// Hauptsimulation
CASE nSimulationStep OF
    0: // Initialisierung
        InitializeSimulation();
        nSimulationStep := 10;
        
    10: // Warte auf Start
        Q_bGrdstlgSchrEinh := TRUE;
        Q_bZustellZylAusgef := FALSE;
        fTiefe := 80.0; // Startposition oben
        
        IF I_bSchraubHub THEN
            nSimulationStep := 20;
            Q_sDebugInfo := 'Zylinder fährt aus';
        END_IF
        
    20: // Zylinder ausfahren
        SimulateZylinder();
        
        IF Q_bZustellZylAusgef THEN
            nSimulationStep := 30;
            Q_sDebugInfo := 'Bereit zum Schrauben';
        END_IF
        
    30: // Schraubvorgang simulieren
        SimulateScrewing();
        
        // Zurück wenn Schraubhub weg
        IF NOT I_bSchraubHub THEN
            nSimulationStep := 40;
        END_IF
        
    40: // Rückfahrt
        SimulateRetraction();
        
        IF Q_bGrdstlgSchrEinh THEN
            nSimulationStep := 10;
        END_IF
END_CASE

// NC-Achsen Simulation updaten
UpdateNCAxes();

// Debug-Ausgänge
Q_fSimTiefe := fTiefe;
Q_fSimDrehmoment := fDrehmoment;
Q_fSimDrehzahl := fDrehzahl;

METHOD PRIVATE CalculateRamp : LREAL
VAR_INPUT
    fActual     : LREAL;    // Aktueller Wert
    fTarget     : LREAL;    // Zielwert
    fRampUp     : LREAL;    // Anstiegsgeschwindigkeit
    fRampDown   : LREAL;    // Abstiegsgeschwindigkeit
END_VAR
// Einfache Rampenberechnung
IF fActual < fTarget THEN
    // Aufwärts
    CalculateRamp := fActual + fRampUp;
    IF CalculateRamp > fTarget THEN
        CalculateRamp := fTarget;
    END_IF
ELSIF fActual > fTarget THEN
    // Abwärts
    CalculateRamp := fActual - fRampDown;
    IF CalculateRamp < fTarget THEN
        CalculateRamp := fTarget;
    END_IF
ELSE
    // Ziel erreicht
    CalculateRamp := fTarget;
END_IF

// Begrenzung auf positive Werte
IF CalculateRamp < 0 THEN
    CalculateRamp := 0;
END_IF
END_METHOD

METHOD InitializeSimulation
VAR
END_VAR
// Simulationsparameter basierend auf gewähltem Fall setzen
CASE I_nSimulatedCase OF
    0: // Normalfall - alles OK
        bSchraubeVorhanden := TRUE;
        bMaterialHart := FALSE;
        bMaterialWeich := FALSE;
        Q_sDebugInfo := 'Simulation: Normalfall';
        
    1: // Fall 1: Negative Toleranz & Drehmoment erreicht
        bSchraubeVorhanden := TRUE;
        bMaterialHart := TRUE;
        bMaterialWeich := FALSE;
        Q_sDebugInfo := 'Simulation: Fall 1 - Hartes Material';
        
    2: // Fall 2: Negative Toleranz & Solltiefe erreicht
        bSchraubeVorhanden := TRUE;
        bMaterialHart := FALSE;
        bMaterialWeich := TRUE;
        Q_sDebugInfo := 'Simulation: Fall 2 - Weiches Material';
        
    3: // Fall 3: Positive Toleranz
        bSchraubeVorhanden := TRUE;
        bMaterialHart := FALSE;
        bMaterialWeich := FALSE;
        Q_sDebugInfo := 'Simulation: Fall 3 - Positive Toleranz';
        
    4: // Fall 4: Keine Schraube
        bSchraubeVorhanden := FALSE;
        bMaterialHart := FALSE;
        bMaterialWeich := FALSE;
        Q_sDebugInfo := 'Simulation: Fall 4 - Keine Schraube';
END_CASE

// Startwerte setzen
fAchsPosition := 0;
fTiefe := 80.0; // Startposition oben
fDrehmoment := 0;
fDrehzahl := 0;
fDrehzahlRampe := 0;
fDrehmomentRampe := 0;

// Rampenparameter setzen
fRampeBeschleunigung := 50.0;  // 50 U/min pro 10ms Zyklus = 5000 U/min/s
fRampeBremsung := 100.0;        // 100 U/min pro 10ms Zyklus = 10000 U/min/s
fDrehmomentAnstieg := 0.02;     // 0.02 Nm pro 10ms Zyklus = 2 Nm/s
END_METHOD

METHOD ResetSimulation
VAR
END_VAR
// Alle Variablen zurücksetzen
fAchsPosition := 0;
fTiefe := 80.0;
fDrehmoment := 0;
fDrehzahl := 0;
fZielDrehzahl := 0;

Q_bZustellZylAusgef := FALSE;
Q_bGrdstlgSchrEinh := TRUE;

nSimulationStep := 0;

// Timer zurücksetzen
tonZylinder(IN:=FALSE);
tonTiefenSimulation(IN:=FALSE);
tonDrehmomentAufbau(IN:=FALSE);

Q_sDebugInfo := 'Simulation zurückgesetzt';
END_METHOD

METHOD SimulateRetraction
VAR
END_VAR
// Rückfahrt simulieren
Q_bZustellZylAusgef := FALSE;

// Tiefe zurückfahren
IF fTiefe < 80.0 THEN
    fTiefe := fTiefe + 1.0; // 1mm pro Zyklus hoch
ELSE
    fTiefe := 80.0;
    Q_bGrdstlgSchrEinh := TRUE;
END_IF

// Drehzahl auf 0
fDrehzahl := 0;
fDrehmoment := 0;

Q_sDebugInfo := 'Rückfahrt in Grundstellung';
END_METHOD

METHOD SimulateScrewing
VAR
    fTiefenGeschwindigkeit : LREAL;
    fDrehmomentZiel : LREAL;
END_VAR
// Drehzahl aus NC-Achse lesen
fZielDrehzahl := arrNcAchsen[I_nAchsId].stAuftrg.fPTP_Geschw * I_fMaxDrehzahl / 100;

// Einfache Drehzahlrampe implementieren
IF fDrehzahl < fZielDrehzahl THEN
    // Beschleunigen
    fDrehzahl := fDrehzahl + fRampeBeschleunigung;
    IF fDrehzahl > fZielDrehzahl THEN
        fDrehzahl := fZielDrehzahl; // Begrenzen auf Zielwert
    END_IF
ELSIF fDrehzahl > fZielDrehzahl THEN
    // Bremsen
    fDrehzahl := fDrehzahl - fRampeBremsung;
    IF fDrehzahl < fZielDrehzahl THEN
        fDrehzahl := fZielDrehzahl; // Begrenzen auf Zielwert
    END_IF
    IF fDrehzahl < 0 THEN
        fDrehzahl := 0; // Nicht negativ werden
    END_IF
END_IF

// Achsposition updaten (Winkel)
IF fDrehzahl > 0 THEN
    fAchsPosition := fAchsPosition + (fDrehzahl / 60 * 360 * 0.01); // 10ms Zykluszeit
END_IF

// Tiefensimulation basierend auf Fall
CASE I_nSimulatedCase OF
    0: // Normalfall
        fTiefenGeschwindigkeit := fDrehzahl / 1000; // Normal
        fDrehmomentZiel := 1.4; // Normales Drehmoment
        
    1: // Hartes Material
        fTiefenGeschwindigkeit := fDrehzahl / 2000; // Langsamer
        fDrehmomentZiel := 1.8; // Hohes Drehmoment
        
    2: // Weiches Material  
        fTiefenGeschwindigkeit := fDrehzahl / 800; // Schneller
        fDrehmomentZiel := 0.5; // Niedriges Drehmoment
        
    3: // Positive Toleranz
        fTiefenGeschwindigkeit := fDrehzahl / 1200;
        fDrehmomentZiel := 1.6;
        
    4: // Keine Schraube
        fTiefenGeschwindigkeit := fDrehzahl / 500; // Sehr schnell
        fDrehmomentZiel := 0.1; // Fast kein Drehmoment
END_CASE

// Tiefe ändern wenn Motor dreht
IF fDrehzahl > 10 AND I_bSchrAuswurf THEN
    IF bSchraubeVorhanden THEN
        // Mit Schraube - normale Geschwindigkeit
        IF fTiefe > I_fSollTiefe THEN
            fTiefe := fTiefe - fTiefenGeschwindigkeit;
            
            // Drehmoment aufbauen je nach Tiefe
            IF fTiefe < (I_fSollTiefe + 5) THEN
                // Kurz vor Ziel - Drehmoment steigt
                tonDrehmomentAufbau(IN:=TRUE, PT:=T#200MS);
                IF tonDrehmomentAufbau.Q OR fDrehmoment < fDrehmomentZiel THEN
                    fDrehmoment := fDrehmoment + fDrehmomentAnstieg;
                END_IF
            END_IF
        ELSE
            // Solltiefe erreicht
            fTiefe := I_fSollTiefe;
        END_IF
    ELSE
        // Ohne Schraube - fährt viel tiefer
        IF fTiefe > (I_fSollTiefe - 15) THEN
            fTiefe := fTiefe - fTiefenGeschwindigkeit * 2;
        END_IF
    END_IF
END_IF

// Drehmoment begrenzen
IF fDrehmoment > I_fMaxDrehmoment THEN
    fDrehmoment := I_fMaxDrehmoment;
END_IF
END_METHOD

METHOD SimulateZylinder
VAR
END_VAR
// Zylinderbewegung simulieren
tonZylinder(IN:=TRUE, PT:=T#500MS);

IF I_bSchrAuswurf THEN
    // Linear nach unten fahren während Auswurf
    IF fTiefe > 10.0 THEN
        fTiefe := fTiefe - 0.5; // 0.5mm pro Zyklus
    ELSE
        fTiefe := 10.0; // Aufsetzhöhe
    END_IF
END_IF

// Nach Timer ist Zylinder ausgefahren
IF tonZylinder.Q THEN
    Q_bZustellZylAusgef := TRUE;
    Q_bGrdstlgSchrEinh := FALSE;
    tonZylinder(IN:=FALSE);
END_IF
END_METHOD

METHOD UpdateNCAxes
VAR
END_VAR
// NC-Achsen-Strukturen mit Simulationswerten füllen
IF I_bSimulationEnable THEN
    
    // Encoder-Position (Tiefe)
    arrNcAchsen[I_nEncId].fPosIstwert := fTiefe;
    
    // Motor-Achse
    arrNcAchsen[I_nAchsId].fPosIstwert := fAchsPosition;
    arrNcAchsen[I_nAchsId].fVeloIstwert := fDrehzahl;
    
    // Drehmoment in 0.1% umrechnen (Annahme: 2Nm = 100%)
    arrNcAchsen[I_nAchsId].stEinAusG.I_nDrehmomentIstwert := LREAL_TO_INT(fDrehmoment / I_fMaxDrehmoment * 1000);
    
    // Status-Bits setzen
    arrNcAchsen[I_nAchsId].stStatus.bInStillst := (fDrehzahl < 1.0);
    arrNcAchsen[I_nAchsId].stStatus.bFaehrtPos := (fDrehzahl > 10.0);
    arrNcAchsen[I_nAchsId].stStatus.bFahrbewAkt := (fDrehzahl > 1.0);
    
    // Betriebsbereit
    arrNcAchsen[I_nAchsId].bBetrbBer := TRUE;
    arrNcAchsen[I_nAchsId].stAuftrg.bPTP_PosiFrg := TRUE;
    
    // Kein Fehler
    arrNcAchsen[I_nAchsId].bNcFehler := FALSE;
    arrNcAchsen[I_nAchsId].stEinAusG.I_nDCStatusword.13 := FALSE;
    
    // Signalstatuswort für Referenzierung
    IF nSimulationStep >= 30 THEN
        arrNcAchsen[I_nAchsId].stEinAusG.I_nSignalstatuswort.0 := TRUE;
    END_IF
    
    // Istwert gesetzt Rückmeldung
    IF arrNcAchsen[I_nAchsId].stGrdfkt.bIstw_setz THEN
        arrNcAchsen[I_nAchsId].stGrdfkt.bIstw_gesetz := TRUE;
    END_IF
    
    // StartAusf Struktur simulieren
    IF arrStartAusf[I_nAchsId].I_bAchseZurArbP THEN
        // Achse läuft
        arrStartAusf[I_nAchsId].Q_bAchseInPos := FALSE;
        arrStartAusf[I_nAchsId].Q_bAchseGestPos := FALSE;
    END_IF
    
    IF arrStartAusf[I_nAchsId].I_bAchseStopPos THEN
        // Achse wurde gestoppt
        arrStartAusf[I_nAchsId].Q_bAchseGestPos := TRUE;
        arrStartAusf[I_nAchsId].Q_bAchseInPos := TRUE;
        fDrehzahl := 0;
    END_IF
    
    // In Position wenn stillsteht
    IF arrNcAchsen[I_nAchsId].stStatus.bInStillst THEN
        arrStartAusf[I_nAchsId].Q_bAchseInPos := TRUE;
    END_IF
END_IF
END_METHOD

END_FUNCTION_BLOCK

// ---- POUs/Simulationsprogramm/PRG_Schrauber_Test.TcPOU
(*
TESTPROGRAMM FÜR SERVOSCHRAUBER MIT SIMULATION
===============================================
Testet alle 4 Schraubfälle und den Normalfall
*)
PROGRAM PRG_Schrauber_Test
VAR
    // Schrauber-Instanz
    fbSchrauber             : FB_Schrauber_PnP_Neu_1;
    
    // Simulation
    fbSimulation            : FB_Schrauber_Simulation;
    
    // Test-Steuerung
    bTestStart              : BOOL;          // Startet einen Testdurchlauf
    bTestStop               : BOOL;          // Stoppt den Test
    nTestCase               : INT := 0;      // Aktueller Testfall (0-4)
    bAutoTest               : BOOL;          // Automatischer Test aller Fälle
    
    // Test-Parameter
    stTestParam             : ST_ParamSKSServoschrauber;
    
    // Hilfsobjekte
    fbObjSchlauch          : FB_Obj_IOSchlauch;
    stMeldung              : ST_MeldServoSchrauber_1;
    
    // Timer für automatischen Test
    tonTestStep            : TON;
    tonTestPause           : TON;
    nAutoTestStep          : INT;
    
    // Ergebnisse
    arrTestResults         : ARRAY[0..4] OF STRING(100);
    bTestRunning           : BOOL;
    sCurrentTest           : STRING(255);
    
    // Bedienung
    bQuittierung           : BOOL;
    bSimulationEnable      : BOOL := TRUE;
    
    // Visualisierung
    fVisTiefe              : LREAL;
    fVisDrehmoment         : LREAL;
    fVisDrehzahl           : LREAL;
    sVisStatus             : STRING(255);
    sVisError              : STRING(255);
END_VAR

// Parameter initialisieren (einmalig)
IF NOT bTestRunning AND stTestParam.fParam_Sollschraubtiefe = 0 THEN
    InitializeTestParameters();
END_IF

// Simulation ausführen
fbSimulation(
    I_bSimulationEnable := bSimulationEnable,
    I_bReset := bTestStop,
    I_nSimulatedCase := nTestCase,
    I_fSollTiefe := stTestParam.fParam_Sollschraubtiefe,
    I_fMaxDrehzahl := 3000,
    I_fMaxDrehmoment := 2.0,
    I_bSchraubHub := fbSchrauber.Q_bSchraubHub,
    I_bSchrAuswurf := fbSchrauber.Q_bSchrAuswurf,
    I_nAchsId := 1,
    I_nEncId := 2
);

// Schrauber-FB aufrufen
fbSchrauber(
    // Steuerungseingänge
    I_bTaktFrg := TRUE,
    I_bTaktStop := bTestStop,
    I_bAuto := TRUE,
    I_bHand := FALSE,
    I_bQuittFehler := bQuittierung,
    I_bGrundstellung := FALSE,
    I_bSchutzbereichOK := fbSimulation.Q_bSchutzbereichOK,
    
    // Prozesseingänge
    I_bTaktStart := bTestStart,
    I_bTaktStartHalb := FALSE,
    I_bGrdstlgSchrEinh := fbSimulation.Q_bGrdstlgSchrEinh,
    I_bZustellZylAusgef := fbSimulation.Q_bZustellZylAusgef,
    
    // Parameter
    I_fSchraubTiefeAuswurf := 80.0,
    I_fTiefentoleranzPos := 1.0,
    I_fTiefentoleranzNeg := 0.5,
    I_nAchsId := 1,
    I_nEncId := 2,
    I_stParam := stTestParam,
    I_tAutoQuit := T#0S,
    
    // Optionale Eingänge
    I_bSchraubeNachschiessen := FALSE,
    I_bReferenzfahrtAktiv := FALSE,
    I_bFreigabeAuswerfen := TRUE,
    I_bSchrauberLogOn := FALSE,
    I_nMotorHersteller := 0,
    I_bHuettenSchr := FALSE,
    
    // In/Out
    IQ_fbObjSchlauch := fbObjSchlauch,
    IQ_stMeldung := stMeldung
);

// Automatischer Test
IF bAutoTest THEN
    AutomaticTestSequence();
ELSE
    nAutoTestStep := 0;
END_IF

// Visualisierungsdaten
UpdateVisualization();

// Testergebnisse speichern
IF fbSchrauber.Q_bDone OR fbSchrauber.Q_bError THEN
    SaveTestResult();
END_IF

METHOD AutomaticTestSequence
VAR
END_VAR
// Automatische Testsequenz durch alle Fälle
CASE nAutoTestStep OF
    0: // Start
        sCurrentTest := 'Automatischer Test gestartet';
        nTestCase := 0;
        nAutoTestStep := 10;
        
    10: // Vorbereitung
        bTestStart := FALSE;
        bQuittierung := FALSE;
        tonTestPause(IN:=TRUE, PT:=T#1S);
        IF tonTestPause.Q THEN
            tonTestPause(IN:=FALSE);
            nAutoTestStep := 20;
        END_IF
        
    20: // Test starten
        sCurrentTest := CONCAT('Teste Fall ', INT_TO_STRING(nTestCase));
        fbObjSchlauch.I_bSchrauberBelegt := TRUE; // Schraube vorhanden
        bTestStart := TRUE;
        nAutoTestStep := 30;
        
    30: // Warten auf Abschluss
        tonTestStep(IN:=TRUE, PT:=T#10S); // Max 10s pro Test
        
        IF fbSchrauber.Q_bDone OR fbSchrauber.Q_bError OR tonTestStep.Q THEN
            tonTestStep(IN:=FALSE);
            bTestStart := FALSE;
            
            // Ergebnis speichern
            IF fbSchrauber.Q_bDone THEN
                arrTestResults[nTestCase] := 'OK';
            ELSIF fbSchrauber.Q_bError THEN
                arrTestResults[nTestCase] := CONCAT('Fehler: ', INT_TO_STRING(fbSchrauber.Q_nErrorId));
            ELSE
                arrTestResults[nTestCase] := 'Timeout';
            END_IF
            
            nAutoTestStep := 40;
        END_IF
        
    40: // Fehler quittieren falls nötig		
        IF fbSchrauber.Q_bError THEN
            bQuittierung := TRUE;
            nAutoTestStep := 50;
        ELSE
            nAutoTestStep := 50;
        END_IF
        
    50: // Nächster Test
        bQuittierung := FALSE;
        tonTestPause(IN:=TRUE, PT:=T#2S);
        
        IF tonTestPause.Q THEN
            tonTestPause(IN:=FALSE);
            
            IF nTestCase < 4 THEN
                nTestCase := nTestCase + 1;
                nAutoTestStep := 10;
            ELSE
                // Alle Tests abgeschlossen
                sCurrentTest := 'Automatischer Test abgeschlossen';
                bAutoTest := FALSE;
                nAutoTestStep := 0;
            END_IF
        END_IF
END_CASE
END_METHOD

METHOD InitializeTestParameters
VAR
END_VAR
// Standard-Testparameter setzen
stTestParam.fParam_Sollschraubtiefe := -5.0;      // Solltiefe 5mm
stTestParam.fParam_SollschraubtiefeHerdumbau := 3.0;
stTestParam.fParam_Umschalttiefe := -3.0;         // Umschalttiefe 3mm
stTestParam.fSchraubTiefeSollDrehzahl := -2.0;    // Solldrehzahl ab 2mm
stTestParam.fParam_Sollmoment := 1.4;             // 1.4 Nm
stTestParam.fParam_Solldrehzahl := 80.0;          // 80% Geschwindigkeit
stTestParam.fStartDrehzahl := 20.0;               // 20% Startgeschwindigkeit

// Zeiten
stTestParam.tParam_ZeitdZustellhubSchr := T#500MS;
stTestParam.tParam_ZeitdSchraubhubSchr := T#1S;
stTestParam.tParam_ZeitdAuswurfSchr := T#500MS;
stTestParam.tParam_ZeitdSchraubTakt := T#3S;

stTestParam.bLogAnwahl := FALSE;
END_METHOD

METHOD SaveTestResult
VAR
    sResult : STRING(100);
END_VAR
// Testergebnis formatieren und speichern
IF fbSchrauber.Q_bDone THEN
    sResult := CONCAT('Fall ', INT_TO_STRING(nTestCase));
    sResult := CONCAT(sResult, ': ERFOLGREICH - Tiefe: ');
    sResult := CONCAT(sResult, LREAL_TO_STRING(fbSimulation.Q_fSimTiefe));
    sResult := CONCAT(sResult, 'mm, Moment: ');
    sResult := CONCAT(sResult, LREAL_TO_STRING(fbSimulation.Q_fSimDrehmoment));
    sResult := CONCAT(sResult, 'Nm');
    
ELSIF fbSchrauber.Q_bError THEN
    sResult := CONCAT('Fall ', INT_TO_STRING(nTestCase));
    sResult := CONCAT(sResult, ': FEHLER ');
    sResult := CONCAT(sResult, INT_TO_STRING(fbSchrauber.Q_nErrorId));
    sResult := CONCAT(sResult, ' - ');
    sResult := CONCAT(sResult, fbSchrauber.Q_sPosZustand);
END_IF

arrTestResults[nTestCase] := sResult;
END_METHOD

METHOD UpdateVisualization
VAR
END_VAR
// Visualisierungsdaten aktualisieren
fVisTiefe := fbSimulation.Q_fSimTiefe;
fVisDrehmoment := fbSimulation.Q_fSimDrehmoment;
fVisDrehzahl := fbSimulation.Q_fSimDrehzahl;

// Status zusammensetzen
sVisStatus := fbSchrauber.Q_sStatus;

IF bAutoTest THEN
    sVisStatus := CONCAT(sVisStatus, ' | ');
    sVisStatus := CONCAT(sVisStatus, sCurrentTest);
END_IF

// Fehleranzeige
IF fbSchrauber.Q_bError THEN
    sVisError := CONCAT('FEHLER ', INT_TO_STRING(fbSchrauber.Q_nErrorId));
    sVisError := CONCAT(sVisError, ': ');
    sVisError := CONCAT(sVisError, fbSchrauber.Q_sPosZustand);
ELSE
    sVisError := 'Kein Fehler';
END_IF

// Test läuft
bTestRunning := fbSchrauber.Q_bBusy;
END_METHOD

END_PROGRAM

// ---- GlobalTextList.TcGTLO
TEXTLIST GlobalTextList
  923 = '%s'
  440 = 'ActPos: %.3f °'
  288 = 'ActPos: %3.f'
  922 = 'ActPos: %3.f °'
  423 = 'ActTiefe: %.3f mm'
  534 = 'ActTiefe: %3.f'
  130 = 'ActTiefe: %3.f mm'
  442 = 'ActTorque: %.3f'
  988 = 'ActTorque: %3.f'
  493 = 'ActVelo: %.3f °/s'
  466 = 'ActVelo: %3.f °/s'
  83 = 'Aktueller Schrauber Status'
  548 = 'Auswurf Start'
  694 = 'Bedienung'
  37 = 'Bedienung Schlauch'
  477 = 'Bedienung Schrauber'
  474 = 'Busy'
  696 = 'Done'
  967 = 'Drehmoment OK'
  998 = 'Error'
  564 = 'Error Drehmoment'
  959 = 'Freigabe'
  309 = 'Letzte Schraube'
  757 = 'Letzter Schraubvorgang'
  771 = 'LetzteTiefe: %3.f mm'
  471 = 'Quit Fehler'
  261 = 'Schlauch Belegt'
  330 = 'Schrauber Belegt'
  515 = 'Status'
  960 = 'Takt Freigabe'
  420 = 'Takt Start'
  772 = 'Takt Stop'
  66 = 'Tiefe: %.3f mm'
  573 = 'Tiefe: %3.f mm'
  53 = 'Tiefe: %3.f °'
  30 = 'Torque: %.3f mm'
  452 = 'Torque: %3.f'
  742 = 'Torque: %3.f mm'
  527 = 'Vereinzelung Start'
  629 = 'Zyl Endlage Grstl'
  191 = 'Zyl Zustell Ausgef'
END_TEXTLIST

// ---- TL_AuswahlSchrauberAblauf.TcTLO
TEXTLIST TL_AuswahlSchrauberAblauf
  0 = 'Reset Ablauf'
  1 = 'Original Ablauf'
  2 = 'Entwickelung Ablauf'
   = ''
END_TEXTLIST

// ---- VISUs/Frame_Schlauch_Bedien.TcVIS
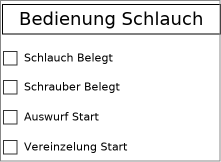
VISUALIZATION Frame_Schlauch_Bedien  // 221x162
VAR_IN_OUT
	bSchlauchBelegt			:BOOL;
	bSchrauberBelegt		:BOOL;
	bAuswurfStart			:BOOL;
	bVereinzelungStart		:BOOL;
END_VAR
    Checkbox (1,72 150x30), "Schrauber Belegt", variable: bSchrauberBelegt
    Checkbox (1,43 150x30), "Schlauch Belegt", variable: bSchlauchBelegt
    Checkbox (1,102 150x30), "Auswurf Start", variable: bAuswurfStart
    Checkbox (1,132 150x30), "Vereinzelung Start", variable: bVereinzelungStart
    Rectangle (2,4 219x30), "Bedienung Schlauch"
END_VISUALIZATION

// ---- VISUs/Frame_Schrauber.TcVIS
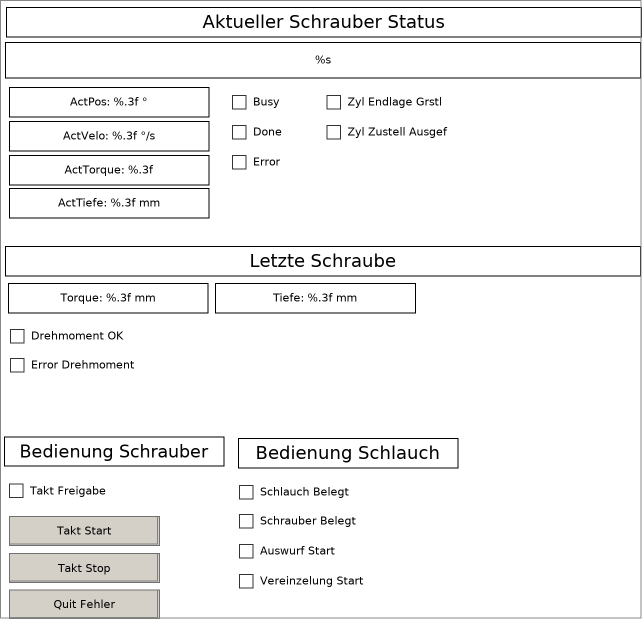
VISUALIZATION Frame_Schrauber  // 642x619
VAR_IN_OUT
	stSKSSchrauberInOut	:ST_SKSSchrauberInOut_Vis;
END_VAR
    Frame (236,434 222x162)
        shows Frame_Schlauch_Bedien(bSchlauchBelegt := stSKSSchrauberInOut.I_bSchlauchBelegt, bSchrauberBelegt := stSKSSchrauberInOut.I_bSchrauberBelegt, bAuswurfStart := stSKSSchrauberInOut.I_bAuswurfStart)
    Frame (2,432 222x187)
        shows Frame_Schrauber_Bedien(bTaktFreigabe := stSKSSchrauberInOut.I_bTaktFrg, bTaktStart := stSKSSchrauberInOut.I_bTaktStart, bTaktStop := stSKSSchrauberInOut.I_bTaktStop, bQuitError := stSKSSchrauberInOut.I_bQuittFehler)
    Frame (3,7 639x373)
        shows Frame_Schrauber_Status(sState := stSKSSchrauberInOut.Q_sStatus, bGrdstlgSchrEinh := stSKSSchrauberInOut.I_bGrdstlgSchrEinh, bZustellZylAusgef := stSKSSchrauberInOut.I_bZustellZylAusgef, bBusy := stSKSSchrauberInOut.Q_bBusy, bDone := stSKSSchrauberInOut.Q_bDone, bError := stSKSSchrauberInOut.Q_bError, bErrorDrehmoment := stSKSSchrauberInOut.Q_bDrehmomentFehler, bDrehmomentOk := stSKSSchrauberInOut.Q_bDrehmomentOk, nDrehmomentMw := stSKSSchrauberInOut.Q_nActTorque, nActPos := stSKSSchrauberInOut.Q_nActPos, nActVelo := stSKSSchrauberInOut.Q_nActVelo, nActTiefe := stSKSSchrauberInOut.Q_nActDepth, nDrehmomentLetzteSchr := stSKSSchrauberInOut.Q_nLastTorque, nTiefeLetzteSchr := stSKSSchrauberInOut.Q_nLastDepth)
END_VISUALIZATION

// ---- VISUs/Frame_Schrauber_Bedien.TcVIS
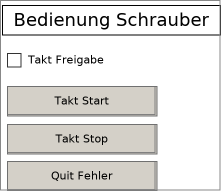
VISUALIZATION Frame_Schrauber_Bedien  // 221x191
VAR_IN_OUT
	bTaktFreigabe	:BOOL;
	bTaktStart		:BOOL;
	bTaktStop		:BOOL;
	bQuitError		:BOOL;
	
END_VAR
    Button (7,124 150x30), "Takt Stop"
        tap bTaktStop
    Button (7,86 150x30), "Takt Start"
        tap bTaktStart
    Checkbox (5,45 150x30), "Takt Freigabe", variable: bTaktFreigabe
    Rectangle (2,5 219x30), "Bedienung Schrauber"
    Button (7,161 150x30), "Quit Fehler"
        tap bQuitError
END_VISUALIZATION

// ---- VISUs/Frame_Schrauber_Status.TcVIS
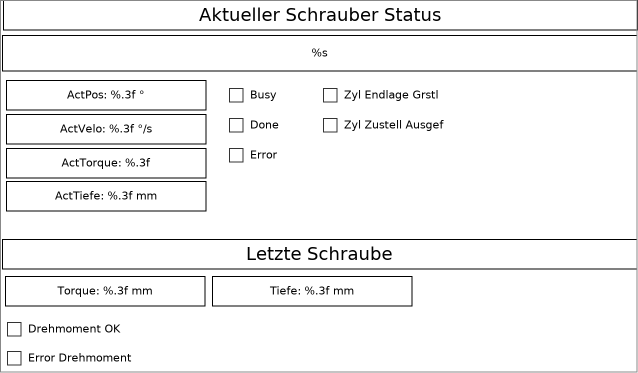
VISUALIZATION Frame_Schrauber_Status  // 638x373
VAR_IN_OUT
	sState	:STRING;
	
	bGrdstlgSchrEinh			: BOOL;
	bZustellZylAusgef			: BOOL;
	
	bBusy	:BOOL;
	bDone	:BOOL;
	bError	:BOOL;
	bErrorDrehmoment		:BOOL;
	bDrehmomentOk			:BOOL;
	nDrehmomentMw			:LREAL;	(* Drehmoment Mittelwert *)
	
	nActPos					:LREAL;
	nActVelo				:LREAL;
	nActTiefe				:LREAL;
	
	nDrehmomentLetzteSchr	:LREAL;	(* Drehmoment Letzte Schraubvorgang *)	
	nTiefeLetzteSchr		:LREAL;	(* Tiefe Letzte Schraubvorgang *)	
END_VAR
    Checkbox (227,80 150x30), "Busy", variable: bBusy, input disabled if: TRUE
    Checkbox (227,110 150x30), "Done", variable: bDone, input disabled if: TRUE
    Checkbox (227,140 150x30), "Error", variable: bError, input disabled if: TRUE
    RoundedRectangle (2,35 635x36), "%s", text variable: sState
    Checkbox (5,314 150x30), "Drehmoment OK", variable: bDrehmomentOk, input disabled if: TRUE
    Rectangle (6,80 200x30), "ActPos: %.3f °", text variable: nActPos
    Rectangle (6,114 200x30), "ActVelo: %.3f °/s", text variable: nActVelo
    Rectangle (6,148 200x30), "ActTorque: %.3f", text variable: nDrehmomentMw
    Rectangle (6,181 200x30), "ActTiefe: %.3f mm", text variable: nActTiefe
    Rectangle (212,276 200x30), "Tiefe: %.3f mm", text variable: nTiefeLetzteSchr
    Rectangle (5,276 200x30), "Torque: %.3f mm", text variable: nDrehmomentLetzteSchr
    Checkbox (5,343 150x30), "Error Drehmoment", variable: bErrorDrehmoment, input disabled if: TRUE
    Rectangle (3,0 635x30), "Aktueller Schrauber Status"
    Rectangle (2,239 635x30), "Letzte Schraube"
    Checkbox (321,80 150x30), "Zyl Endlage Grstl", variable: bGrdstlgSchrEinh, input disabled if: true
    Checkbox (321,110 150x30), "Zyl Zustell Ausgef", variable: bZustellZylAusgef, input disabled if: true
END_VISUALIZATION

// ---- VISUs/Schrauber_Aufruf.TcVIS
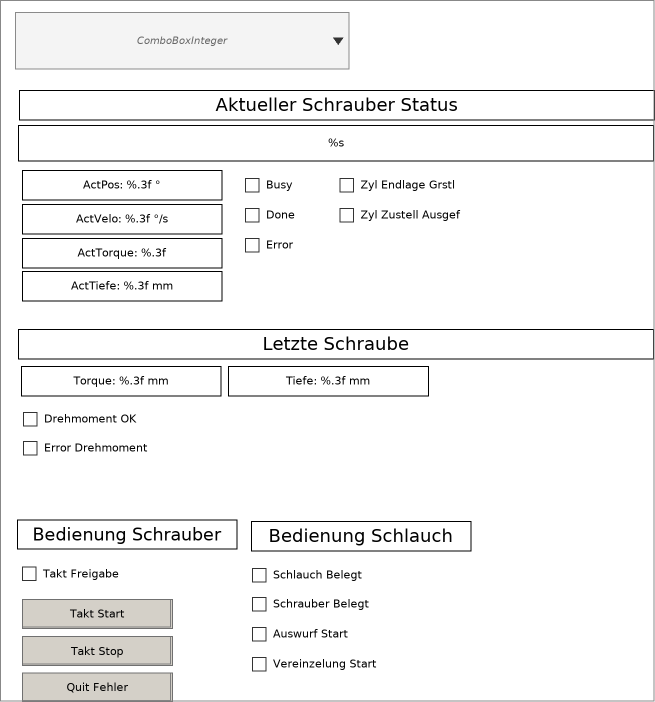
VISUALIZATION Schrauber_Aufruf  // 655x702
    Frame (13,83 642x619)
        shows Frame_Schrauber(stSKSSchrauberInOut := stSKSSchrauberInOut_Vis_Schr_1)
    ComboBoxInteger (15,12 334x57), variable: PRG_Schrauber.iAuswSchrauberMode, text list: 'TL_AuswahlSchrauberAblauf'
END_VISUALIZATION
